(* IEC 61131-3 sources: volt/packages/volt-lsp-iec/test-corpus/lenze-mid/Device/Plc Logic/Application/Library Manager/CAA Types, 80 files *)

(* ---- COUNT.dut ---- *)
TYPE COUNT : __UXINT;
END_TYPE

(* ---- DURATION.dut ---- *)
TYPE DURATION : TIME;
END_TYPE

(* ---- ENDIANESS.dut ---- *)
TYPE ENDIANESS :
(
	UNKNOWN,
	LITTLE,
	BIG
);
END_TYPE

(* ---- ERROR.dut ---- *)
TYPE ERROR :
(
	NO_ERROR
);
END_TYPE

(* ---- FILENAME.dut ---- *)
TYPE FILENAME : STRING(255);
END_TYPE

(* ---- FLOAT.dut ---- *)
TYPE FLOAT : LREAL;
END_TYPE

(* ---- HANDLE.dut ---- *)
TYPE HANDLE : __XWORD;
END_TYPE

(* ---- IDENT.dut ---- *)
TYPE IDENT : DWORD;
END_TYPE

(* ---- PVOID.dut ---- *)
TYPE PVOID : __XWORD;
END_TYPE

(* ---- SIGNED.dut ---- *)
TYPE SIGNED : INT;
END_TYPE

(* ---- SIZE.dut ---- *)
TYPE SIZE : __UXINT;
END_TYPE

(* ---- SYSTYPE.dut ---- *)
TYPE SYSTYPE :
(
	UNKNOWN,
	SMALL,
	MEDIUM,
	LARGE
);
END_TYPE

(* ---- TICK.dut ---- *)
TYPE TICK : __UXINT;
END_TYPE

(* ---- UNSIGNED.dut ---- *)
TYPE UNSIGNED : UINT;
END_TYPE

(* ---- ARCHITECTURE.gvl ---- *)
VAR_GLOBAL
	G_EENDIANESS : ENDIANESS := CalcEndianess();
	G_ESYSTYPE : SYSTYPE := CalcSystemType();
END_VAR

(* ---- CONSTANTS.gvl ---- *)
VAR_GLOBAL
	GC_HINVALID : HANDLE := 0;
	GC_PNULL : PVOID := 0;
	GC_SZZERO : SIZE := 0;
	GC_CTMAX_COUNT : COUNT := -1;
	GC_IDMAX_IDENT : IDENT := -1;
END_VAR

(* ---- SYSTEM.gvl ---- *)
VAR_GLOBAL
	GC_EENDIANESS : ENDIANESS := ENDIANESS.LITTLE;
	GC_ESYSTYPE : SYSTYPE := SYSTYPE.MEDIUM;
END_VAR

(* ---- VERSIONCONSTANTS.gvl ---- *)
VAR_GLOBAL
	GC_BYVERSION : BYTE := 1;
	GC_VERSION_1 : BYTE := 0;
END_VAR

(* ---- CALCENDIANESS.pou ---- *)
FUNCTION CALCENDIANESS : ENDIANESS
END_FUNCTION

(* ---- CALCSYSTEMTYPE.pou ---- *)
FUNCTION CALCSYSTEMTYPE : SYSTYPE
END_FUNCTION

(* ---- COUNT_TO_UDINT.pou ---- *)
FUNCTION COUNT_TO_UDINT : UDINT
VAR_INPUT
	CTVALUE : COUNT;
END_VAR
END_FUNCTION

(* ---- COUNT_TO_UINT.pou ---- *)
FUNCTION COUNT_TO_UINT : UINT
VAR_INPUT
	CTVALUE : COUNT;
END_VAR
END_FUNCTION

(* ---- COUNT_TO_ULINT.pou ---- *)
FUNCTION COUNT_TO_ULINT : ULINT
VAR_INPUT
	CTVALUE : COUNT;
END_VAR
END_FUNCTION

(* ---- DINT_TO_SIGNED.pou ---- *)
FUNCTION DINT_TO_SIGNED : SIGNED
VAR_INPUT
	DIVALUE : DINT;
END_VAR
END_FUNCTION

(* ---- DURATION_TO_LTIME.pou ---- *)
FUNCTION DURATION_TO_LTIME : LTIME
VAR_INPUT
	DURVALUE : DURATION;
END_VAR
END_FUNCTION

(* ---- DURATION_TO_TIME.pou ---- *)
FUNCTION DURATION_TO_TIME : TIME
VAR_INPUT
	DURVALUE : DURATION;
END_VAR
END_FUNCTION

(* ---- DWORD_TO_HANDLE.pou ---- *)
FUNCTION DWORD_TO_HANDLE : HANDLE
VAR_INPUT
	DWVALUE : DWORD;
END_VAR
END_FUNCTION

(* ---- DWORD_TO_IDENT.pou ---- *)
FUNCTION DWORD_TO_IDENT : IDENT
VAR_INPUT
	DWVALUE : DWORD;
END_VAR
END_FUNCTION

(* ---- DWORD_TO_PVOID.pou ---- *)
FUNCTION DWORD_TO_PVOID : PVOID
VAR_INPUT
	DWVALUE : DWORD;
END_VAR
END_FUNCTION

(* ---- FLOAT_TO_LREAL.pou ---- *)
FUNCTION FLOAT_TO_LREAL : LREAL
VAR_INPUT
	FLTVALUE : FLOAT;
END_VAR
END_FUNCTION

(* ---- FLOAT_TO_REAL.pou ---- *)
FUNCTION FLOAT_TO_REAL : REAL
VAR_INPUT
	FLTVALUE : FLOAT;
END_VAR
END_FUNCTION

(* ---- GETSUPPLIERVERSION.pou ---- *)
FUNCTION GETSUPPLIERVERSION : WORD
VAR_INPUT
	XDUMMY : BOOL;
END_VAR
END_FUNCTION

(* ---- HANDLE_TO_DWORD.pou ---- *)
FUNCTION HANDLE_TO_DWORD : DWORD
VAR_INPUT
	HVALUE : HANDLE;
END_VAR
END_FUNCTION

(* ---- HANDLE_TO_LWORD.pou ---- *)
FUNCTION HANDLE_TO_LWORD : LWORD
VAR_INPUT
	HVALUE : HANDLE;
END_VAR
END_FUNCTION

(* ---- HANDLE_TO_WORD.pou ---- *)
FUNCTION HANDLE_TO_WORD : WORD
VAR_INPUT
	HVALUE : HANDLE;
END_VAR
END_FUNCTION

(* ---- IDENT_TO_DWORD.pou ---- *)
FUNCTION IDENT_TO_DWORD : DWORD
VAR_INPUT
	IDVALUE : IDENT;
END_VAR
END_FUNCTION

(* ---- IDENT_TO_WORD.pou ---- *)
FUNCTION IDENT_TO_WORD : WORD
VAR_INPUT
	IDVALUE : IDENT;
END_VAR
END_FUNCTION

(* ---- INT_TO_SIGNED.pou ---- *)
FUNCTION INT_TO_SIGNED : SIGNED
VAR_INPUT
	IVALUE : INT;
END_VAR
END_FUNCTION

(* ---- LINT_TO_SIGNED.pou ---- *)
FUNCTION LINT_TO_SIGNED : SIGNED
VAR_INPUT
	LIVALUE : LINT;
END_VAR
END_FUNCTION

(* ---- LREAL_TO_FLOAT.pou ---- *)
FUNCTION LREAL_TO_FLOAT : FLOAT
VAR_INPUT
	LRVALUE : LREAL;
END_VAR
END_FUNCTION

(* ---- LTIME_TO_DURATION.pou ---- *)
FUNCTION LTIME_TO_DURATION : DURATION
VAR_INPUT
	LTVALUE : LTIME;
END_VAR
END_FUNCTION

(* ---- LWORD_TO_HANDLE.pou ---- *)
FUNCTION LWORD_TO_HANDLE : HANDLE
VAR_INPUT
	LWVALUE : LWORD;
END_VAR
END_FUNCTION

(* ---- LWORD_TO_PVOID.pou ---- *)
FUNCTION LWORD_TO_PVOID : PVOID
VAR_INPUT
	LWVALUE : LWORD;
END_VAR
END_FUNCTION

(* ---- PVOID_TO_DWORD.pou ---- *)
FUNCTION PVOID_TO_DWORD : DWORD
VAR_INPUT
	PVALUE : PVOID;
END_VAR
END_FUNCTION

(* ---- PVOID_TO_LWORD.pou ---- *)
FUNCTION PVOID_TO_LWORD : LWORD
VAR_INPUT
	PVALUE : PVOID;
END_VAR
END_FUNCTION

(* ---- PVOID_TO_WORD.pou ---- *)
FUNCTION PVOID_TO_WORD : WORD
VAR_INPUT
	PVALUE : PVOID;
END_VAR
END_FUNCTION

(* ---- REAL_TO_FLOAT.pou ---- *)
FUNCTION REAL_TO_FLOAT : FLOAT
VAR_INPUT
	RVALUE : REAL;
END_VAR
END_FUNCTION

(* ---- RESMANINCHARGE.pou ---- *)
FUNCTION RESMANINCHARGE : BOOL
VAR_INPUT
	XDUMMY : BOOL;
END_VAR
END_FUNCTION

(* ---- SIGNED_TO_DINT.pou ---- *)
FUNCTION SIGNED_TO_DINT : DINT
VAR_INPUT
	SGNVALUE : SIGNED;
END_VAR
END_FUNCTION

(* ---- SIGNED_TO_INT.pou ---- *)
FUNCTION SIGNED_TO_INT : INT
VAR_INPUT
	SGNVALUE : SIGNED;
END_VAR
END_FUNCTION

(* ---- SIGNED_TO_LINT.pou ---- *)
FUNCTION SIGNED_TO_LINT : LINT
VAR_INPUT
	SGNVALUE : SIGNED;
END_VAR
END_FUNCTION

(* ---- SIZE_TO_UDINT.pou ---- *)
FUNCTION SIZE_TO_UDINT : UDINT
VAR_INPUT
	SZVALUE : SIZE;
END_VAR
END_FUNCTION

(* ---- SIZE_TO_UINT.pou ---- *)
FUNCTION SIZE_TO_UINT : UINT
VAR_INPUT
	SZVALUE : SIZE;
END_VAR
END_FUNCTION

(* ---- SIZE_TO_ULINT.pou ---- *)
FUNCTION SIZE_TO_ULINT : ULINT
VAR_INPUT
	SZVALUE : SIZE;
END_VAR
END_FUNCTION

(* ---- TASKLOCK.pou ---- *)
FUNCTION TASKLOCK : ERROR
VAR_INPUT
	XDUMMY : BOOL;
END_VAR
END_FUNCTION

(* ---- TASKUNLOCK.pou ---- *)
FUNCTION TASKUNLOCK : ERROR
VAR_INPUT
	XDUMMY : BOOL;
END_VAR
END_FUNCTION

(* ---- TICK_TO_UDINT.pou ---- *)
FUNCTION TICK_TO_UDINT : UDINT
VAR_INPUT
	TKVALUE : TICK;
END_VAR
END_FUNCTION

(* ---- TICK_TO_UINT.pou ---- *)
FUNCTION TICK_TO_UINT : UINT
VAR_INPUT
	TKVALUE : TICK;
END_VAR
END_FUNCTION

(* ---- TICK_TO_ULINT.pou ---- *)
FUNCTION TICK_TO_ULINT : ULINT
VAR_INPUT
	TKVALUE : TICK;
END_VAR
END_FUNCTION

(* ---- TIME_TO_DURATION.pou ---- *)
FUNCTION TIME_TO_DURATION : DURATION
VAR_INPUT
	TVALUE : TIME;
END_VAR
END_FUNCTION

(* ---- UDINT_TO_COUNT.pou ---- *)
FUNCTION UDINT_TO_COUNT : COUNT
VAR_INPUT
	UDIVALUE : UDINT;
END_VAR
END_FUNCTION

(* ---- UDINT_TO_SIZE.pou ---- *)
FUNCTION UDINT_TO_SIZE : SIZE
VAR_INPUT
	UDIVALUE : UDINT;
END_VAR
END_FUNCTION

(* ---- UDINT_TO_TICK.pou ---- *)
FUNCTION UDINT_TO_TICK : TICK
VAR_INPUT
	UDIVALUE : UDINT;
END_VAR
END_FUNCTION

(* ---- UDINT_TO_UNSIGNED.pou ---- *)
FUNCTION UDINT_TO_UNSIGNED : UNSIGNED
VAR_INPUT
	UDIVALUE : UDINT;
END_VAR
END_FUNCTION

(* ---- UINT_TO_COUNT.pou ---- *)
FUNCTION UINT_TO_COUNT : COUNT
VAR_INPUT
	UIVALUE : UINT;
END_VAR
END_FUNCTION

(* ---- UINT_TO_SIZE.pou ---- *)
FUNCTION UINT_TO_SIZE : SIZE
VAR_INPUT
	UIVALUE : UINT;
END_VAR
END_FUNCTION

(* ---- UINT_TO_TICK.pou ---- *)
FUNCTION UINT_TO_TICK : TICK
VAR_INPUT
	UIVALUE : UINT;
END_VAR
END_FUNCTION

(* ---- UINT_TO_UNSIGNED.pou ---- *)
FUNCTION UINT_TO_UNSIGNED : UNSIGNED
VAR_INPUT
	UIVALUE : UINT;
END_VAR
END_FUNCTION

(* ---- ULINT_TO_COUNT.pou ---- *)
FUNCTION ULINT_TO_COUNT : COUNT
VAR_INPUT
	ULIVALUE : ULINT;
END_VAR
END_FUNCTION

(* ---- ULINT_TO_SIZE.pou ---- *)
FUNCTION ULINT_TO_SIZE : SIZE
VAR_INPUT
	ULIVALUE : ULINT;
END_VAR
END_FUNCTION

(* ---- ULINT_TO_TICK.pou ---- *)
FUNCTION ULINT_TO_TICK : TICK
VAR_INPUT
	ULIVALUE : ULINT;
END_VAR
END_FUNCTION

(* ---- ULINT_TO_UNSIGNED.pou ---- *)
FUNCTION ULINT_TO_UNSIGNED : UNSIGNED
VAR_INPUT
	ULIVALUE : ULINT;
END_VAR
END_FUNCTION

(* ---- UNSIGNED_TO_UDINT.pou ---- *)
FUNCTION UNSIGNED_TO_UDINT : UDINT
VAR_INPUT
	USGVALUE : UNSIGNED;
END_VAR
END_FUNCTION

(* ---- UNSIGNED_TO_UINT.pou ---- *)
FUNCTION UNSIGNED_TO_UINT : UINT
VAR_INPUT
	USGVALUE : UNSIGNED;
END_VAR
END_FUNCTION

(* ---- UNSIGNED_TO_ULINT.pou ---- *)
FUNCTION UNSIGNED_TO_ULINT : ULINT
VAR_INPUT
	USGVALUE : UNSIGNED;
END_VAR
END_FUNCTION

(* ---- WORD_TO_HANDLE.pou ---- *)
FUNCTION WORD_TO_HANDLE : HANDLE
VAR_INPUT
	WVALUE : WORD;
END_VAR
END_FUNCTION

(* ---- WORD_TO_IDENT.pou ---- *)
FUNCTION WORD_TO_IDENT : IDENT
VAR_INPUT
	WVALUE : WORD;
END_VAR
END_FUNCTION

(* ---- WORD_TO_PVOID.pou ---- *)
FUNCTION WORD_TO_PVOID : PVOID
VAR_INPUT
	WVALUE : WORD;
END_VAR
END_FUNCTION

(* ---- BOLT.pou ---- *)
FUNCTION_BLOCK BOLT
VAR
	UDISYNC : UDINT := 0;
	CTSTATE : COUNT := 0;
	CTRESERVED : COUNT := 0;
	XFREE : BOOL := TRUE;
END_VAR
END_FUNCTION_BLOCK

METHOD FREE : BOOL
END_METHOD

METHOD RESERVE : BOOL
VAR_IN_OUT
	CTVALUE : COUNT;
END_VAR
END_METHOD

METHOD LEAVE : BOOL
END_METHOD

METHOD ENTER : BOOL
END_METHOD

(* ---- SEMA.pou ---- *)
FUNCTION_BLOCK SEMA
VAR_INPUT
	CTPRESET : COUNT := 1;
END_VAR
VAR
	UDISYNC : UDINT := 0;
	CTSTATE : COUNT := 1;
	PRESET : COUNT;
END_VAR
END_FUNCTION_BLOCK

METHOD REQUEST : BOOL
END_METHOD

METHOD RELEASE : BOOL
END_METHOD

METHOD INIT
END_METHOD
